{attribute 'hide'}
FUNCTION_BLOCK ABSTRACT FB_StatusExecuteFB
VAR_INPUT
END_VAR
VAR_OUTPUT
END_VAR
VAR
	bExecute						: BOOL;
	bBusy							: BOOL;
	bCommandAborted					: BOOL;
	bDone							: BOOL;
	bError							: BOOL;
	udiErrorID						: UDINT;
END_VAR

//{warning 'add method implementation '}
METHOD ABSTRACT METH_Busy : BOOL
END_METHOD

//{warning 'add method implementation '}
METHOD PROTECTED METH_CommandAborted : BOOL
Prop_CommandAborted := TRUE;
Prop_Busy := FALSE;
END_METHOD

//{warning 'add method implementation '}
METHOD PROTECTED METH_Done : BOOL
Prop_Done := TRUE;
Prop_Busy := FALSE;
END_METHOD

METHOD ABSTRACT METH_Enter : BOOL
VAR_INPUT
END_VAR
END_METHOD

//{warning 'add method implementation '}
METHOD PROTECTED METH_Error : BOOL
Prop_Error := TRUE;
Prop_Busy := FALSE;
END_METHOD

//{warning 'add method implementation '}
METHOD PROTECTED METH_Execute : BOOL
Prop_Execute := TRUE;
Prop_Busy := TRUE;
END_METHOD

METHOD ABSTRACT METH_Exit : BOOL
VAR_INPUT
END_VAR
END_METHOD

METHOD ABSTRACT METH_Main : BOOL
VAR_INPUT
END_VAR
END_METHOD

{warning 'add property implementation'}
PROPERTY Prop_Busy : BOOL
GET
Prop_Busy := bBusy;
END_GET
SET
bBusy := Prop_Busy;
END_SET
END_PROPERTY

{warning 'add property implementation'}
PROPERTY Prop_CommandAborted : BOOL
GET
Prop_CommandAborted := bCommandAborted;
END_GET
SET
bCommandAborted := Prop_CommandAborted;
END_SET
END_PROPERTY

{warning 'add property implementation'}
PROPERTY Prop_Done : BOOL
GET
Prop_Done := bDone;
END_GET
SET
bDone := Prop_Done;
END_SET
END_PROPERTY

{warning 'add property implementation'}
PROPERTY Prop_Error : BOOL
GET
Prop_Error := bError;
END_GET
SET
bError := Prop_Error;
END_SET
END_PROPERTY

{warning 'add property implementation'}
PROPERTY Prop_ErrorID : UDINT
GET
Prop_ErrorID := udiErrorID;
END_GET
SET
udiErrorID := Prop_ErrorID;
END_SET
END_PROPERTY

{warning 'add property implementation'}
PROPERTY Prop_Execute : BOOL
GET
Prop_Execute := bExecute;
END_GET
SET
bExecute := Prop_Execute;
END_SET
END_PROPERTY

END_FUNCTION_BLOCK

(* stored: Version 1.1.0.1, ProductVersion 3.1.4024.12
   POU FB_StatusExecuteFB: Id {d5f257bd-48dd-4936-96a9-f8db7aae2619}, SpecialFunc None
   Method METH_Busy: Id {e4701e2b-57b4-45d2-856e-6a77476b5fa3}
   Method METH_CommandAborted: Id {8a06b7e9-cd23-4ca9-8366-3af741ea5757}
   Method METH_Done: Id {27acebb5-47cc-4300-80a1-d92566086c17}
   Method METH_Enter: Id {b065b700-5499-485c-a7d4-22501d5dac27}
   Method METH_Error: Id {4884cb9b-c09d-440b-91cb-bbf4984ee557}
   Method METH_Execute: Id {ca35221a-7db9-428d-afe1-aeeda118cf30}
   Method METH_Exit: Id {43f1cf57-ff0a-40a4-b771-62f5990519e7}
   Method METH_Main: Id {b81c8b24-0878-4853-9aa3-372995571ff9}
   Property Prop_Busy: Id {78d901d9-e32d-4c7c-b069-3904cfbff611}
   Get Get: Id {c1edb156-2f97-4178-a03c-871734dd572a}
   Set Set: Id {05a8f90d-af7c-4a39-95cd-eddfa3e33f26}
   Property Prop_CommandAborted: Id {5122f78b-f476-4fb1-884d-61606e780032}
   Get Get: Id {4daf0701-d5ec-4649-ad81-255fd0f21a07}
   Set Set: Id {c0a05eb2-27e6-49a0-9c22-b070ea7a90f0}
   Property Prop_Done: Id {3d18b7c5-0a69-449e-9562-bfc631b13a0d}
   Get Get: Id {d9f8d2f1-f519-4aee-acad-ebd3b2aa6003}
   Set Set: Id {24565ebb-385c-4d4d-a78b-7134384063ed}
   Property Prop_Error: Id {3580ffba-c3f3-4488-ade4-ce95f2dc0c4c}
   Get Get: Id {2ce8b1f1-0fbc-49b4-905a-6f1d6ce087b9}
   Set Set: Id {8e9412eb-df20-4fc2-966b-c6cff64d4003}
   Property Prop_ErrorID: Id {a6317e23-c332-4094-8c03-55f6a312fcb4}
   Get Get: Id {d7f86459-134e-4f7c-8527-53add93dbe92}
   Set Set: Id {cd21a140-ab88-4a6a-913b-3fe8e00e6966}
   Property Prop_Execute: Id {a8301cd7-a733-4882-9e6e-d6eb755bae5c}
   Get Get: Id {109fc49f-50f7-45f4-8d58-62ac2daea40c}
   Set Set: Id {a16a2442-d7dd-436b-aca9-da84d57563f9} *)
